Fanuc KAREL source: kf00070.KL

PROGRAM KF00070
%STACKSIZE=65535
%PRIORITY=65535
%NOLOCKGROUP
VAR
I : INTEGER
J : INTEGER
X : REAL
Y : REAL
B : BOOLEAN
C : BOOLEAN
TXT : STRING[80]
TXT2 : STRING[80]
AI : ARRAY[4] OF INTEGER
BI : ARRAY[4] OF INTEGER
P : XYZWPR
JP : JOINTPOS9
PF : POSITION
V1 : VECTOR
V2 : VECTOR
STATUS : INTEGER
BEGIN
TXT='12'
TXT2='2'
I=12
X=2.5
-- UNSAFE_SOURCE_IR line 25: I = native_s16_value(AI)
END KF00070
